INTERFACE I_XTS_Trigger  EXTENDS I_CH_Object

{attribute 'monitoring':='call'}
PROPERTY HR : HRESULT
GET
END_GET
END_PROPERTY

PROPERTY ListOfMoversToCheck : I_CH_List
SET
END_SET
END_PROPERTY

{attribute 'monitoring':='call'}
PROPERTY MoverAtTrigger : I_XTS_Mover
GET
END_GET
END_PROPERTY

{attribute 'monitoring':='call'}
PROPERTY MoverDetected : BOOL
GET
END_GET
END_PROPERTY

{attribute 'monitoring':='call'}
PROPERTY PositionOnTrack : LREAL
GET
END_GET
SET
END_SET
END_PROPERTY

{attribute 'monitoring':='call'}
PROPERTY TimeStamp : T_DCTIME64;
GET
END_GET
END_PROPERTY

{attribute 'monitoring':='call'}
PROPERTY TriggerDirection : Tc2_MC2.MC_Direction
GET
END_GET
SET
END_SET
END_PROPERTY

END_INTERFACE

(* stored: Version 1.1.0.1, ProductVersion 3.1.4024.12
   Itf I_XTS_Trigger: Id {397858f5-d03c-4a61-80a2-99e2e9a15f03}
   Property HR: Id {ee86a53c-863d-4cb1-945a-719afaee9193}
   Get Get: Id {7386810f-eca8-4bd1-9276-fcc98215ccd8}
   Property ListOfMoversToCheck: Id {d0696dd1-ec69-4f6e-911b-ce8e251538d6}
   Set Set: Id {049c481b-a11e-4754-ad00-b7b3d8ac8249}
   Property MoverAtTrigger: Id {79b21152-3f8e-411d-8737-5e86b4875174}
   Get Get: Id {a6ac075a-345c-425b-bfd2-6f3067a58455}
   Property MoverDetected: Id {ba0c50c9-9bc8-44a5-98f4-9433ef35f31a}
   Get Get: Id {159bb0f2-496f-439c-8f32-c4783e326f15}
   Property PositionOnTrack: Id {f6c0903c-8316-4146-a5df-eb5c54641ed0}
   Get Get: Id {0de141bc-92f3-49f5-90b0-e2fe230225ef}
   Set Set: Id {5f6f914c-cc07-4113-91dc-ddb5827fa663}
   Property TimeStamp: Id {d0533e2f-0608-43d0-80d9-f762342157b4}
   Get Get: Id {11b40524-060e-47f8-8962-af1c7c26a318}
   Property TriggerDirection: Id {018277f0-84fb-4720-9b55-07c191e35504}
   Get Get: Id {3b889148-5f62-4ea9-88c1-e58f96900af7}
   Set Set: Id {36e70e54-a41b-425c-acef-33e2619ed5b0} *)
